(* IEC 61131-3 sources: lacyccom/src/Blocks/Drives (part 2) *)

(* ---- classRtcSinamics.st ---- *)
USING Siemens.Simatic.Clocks;
USING System.DateTime;

NAMESPACE Simatic.Ax.LAcycCom
    CLASS LAcycCom_classRtcSinamics
        VAR
            statrtcRealTimeSyncPING         : BOOL;
            statRetSetrtcRealTimeSyncPING   : BOOL;
            statRetResetrtcRealTimeSyncPING : BOOL;
            statrequestBuffer               : Resourcemanager;
            statWriteDrivePara              : LAcycCom_classWriteDriveSingleParams;
            statFBState                     : LAcycCom_ReadWriteStatus := LAcycCom_ReadWriteStatus#FB_IDLE;   // States in the function block state machine
            statFBSubState                  : LAcycCom_ReadWriteStatus := LAcycCom_ReadWriteStatus#FB_BUSY_PING;   // States in the function block during processing (busy state)
            statStatus                      : WORD := STATUS_NO_CALL;   // Static value for output status
            statStateNumber                 : LAcycCom_ReadWriteStatus;   // State of the FB when error occurred
            stathardwareId                  : HW_IO;
            statsystemDateTime              : LDATE_AND_TIME;
            statWritepara                   : LAcycCom_classWriteDriveSingleParams;
            statactmilisecond               : DWORD;
            statexternTime                  : BOOL;
            StatEnablePing                  : BOOL;
        END_VAR

        VAR CONSTANT
            STATUS_EXECUTION_FINISHED   : WORD := WORD#16#0000;   // Execution finished without errors
            STATUS_NO_CALL              : WORD := WORD#16#7000;   // No call of FB
            STATUS_ALLOCATE             : WORD := WORD#16#7001;   // FB is currently allocating a request element
            STATUS_GET_RESOURCE         : WORD := WORD#16#7002;   // FB is waiting until it has “speaking rights”
            STATUS_BUSY                 : WORD := WORD#16#7003;   // FB is currently in processing
            STATUS_RELEASE              : WORD := WORD#16#7004;   // FB is releasing the allocated element
            ERR_UNDEFINED_STATE         : WORD := WORD#16#8611;   // Error due to an undefined state
        END_VAR

        METHOD PUBLIC execute

            IF NOT (statFBState = LAcycCom_ReadWriteStatus#FB_IDLE OR
                statFBState = LAcycCom_ReadWriteStatus#FB_DONE OR
                statFBState = LAcycCom_ReadWriteStatus#FB_ERROR ) THEN  // Functionality running
                CASE statFBState OF
                    LAcycCom_ReadWriteStatus#FB_FIRST_CYCLE:  // First cycle state

                        This.FIRST_CYCLE();

                    LAcycCom_ReadWriteStatus#FB_BUSY:

                        This.BUSY();

                    ELSE
                    statStatus := ERR_UNDEFINED_STATE;
                    statStateNumber := statFBState;
                    statFBState := LAcycCom_ReadWriteStatus#FB_ERROR;
                END_CASE;
            END_IF;

        END_METHOD

        Method Private FIRST_CYCLE

            statrtcRealTimeSyncPING         := FALSE;
            statRetSetrtcRealTimeSyncPING   := FALSE;
            statRetResetrtcRealTimeSyncPING := FALSE;

            statFBState     := LAcycCom_ReadWriteStatus#FB_BUSY;
            statFBSubState  := LAcycCom_ReadWriteStatus#FB_BUSY_PING_RESET;
        END_METHOD

        Method PRIVATE Busy
            VAR
                actDays         : INT;
                actMonth        : INT;
                actYear         : INT;
                actHour         : INT;
                actMinute       : INT;
                actSecond       : INT;
                actMillisecond  : INT;
                elapsedYears    : INT;
                elapsedDays     : DINT;
                loop            : DINT;
            END_VAR

            CASE statFBSubState OF
                LAcycCom_ReadWriteStatus#FB_BUSY_PING_RESET:
                    IF statRetResetrtcRealTimeSyncPING THEN
                        statFBSubState := LAcycCom_ReadWriteStatus#FB_BUSY_WRREC;

                        statWriteDrivePara.execute();
                        statWriteDrivePara.Start(driveObjectId  := UINT#1,   // Optional: Identification number of the drive object (value =0: driveObjectId is NOT used, i.e. the corresponding drive object is only addressed via the hardwareId)
                                                hardwareId      := stathardwareId,   // Hardware identifier of the hardware module
                                                parameterNumber := UINT#3100,   // Number of the parameter
                                                index           := UINT#0,   // Parameter index
                                                value           := REAL#1.0,
                                                dwValue         := DWORD#0
                                                );
                    END_IF;

                LAcycCom_ReadWriteStatus#FB_BUSY_WRREC:
                    statWriteDrivePara.execute();

                    IF  statWriteDrivePara.Status() = LAcycComstateDef#DONE THEN
                        statFBSubState := LAcycCom_ReadWriteStatus#FB_BUSY_WRREC_1;
                        IF StatEnablePing THEN
                            statWriteDrivePara.Start(driveObjectId  := UINT#1,   // Optional: Identification number of the drive object (value =0: driveObjectId is NOT used, i.e. the corresponding drive object is only addressed via the hardwareId)
                                                    hardwareId      := stathardwareId,   // Hardware identifier of the hardware module
                                                    parameterNumber := UINT#3103,   // Number of the parameter
                                                    index           := UINT#0,   // Parameter index
                                                    value           := REAL#0.0,
                                                    dwValue         := DWORD#0
                                                    );
                        ELSE
                            statWriteDrivePara.Start(driveObjectId  := UINT#1,   // Optional: Identification number of the drive object (value =0: driveObjectId is NOT used, i.e. the corresponding drive object is only addressed via the hardwareId)
                                                    hardwareId      := stathardwareId,   // Hardware identifier of the hardware module
                                                    parameterNumber := UINT#3103,   // Number of the parameter
                                                    index           := UINT#0,   // Parameter index
                                                    value           := REAL#2.0,
                                                    dwValue         := DWORD#0
                                                    );
                        END_IF;
                    END_IF;

                LAcycCom_ReadWriteStatus#FB_BUSY_WRREC_1:
                    statWriteDrivePara.execute();

                    IF  statWriteDrivePara.Status() = LAcycComstateDef#DONE THEN
                        statFBSubState := LAcycCom_ReadWriteStatus#FB_BUSY_PING;
                    END_IF;

                LAcycCom_ReadWriteStatus#FB_BUSY_PING:
                    statrtcRealTimeSyncPING := StatEnablePing;
                    IF statRetSetrtcRealTimeSyncPING OR NOT StatEnablePing THEN

                        IF NOT statexternTime THEN
                            GetSystemDateTime(value => statsystemDateTime);
                        END_IF;

                        SplitDateAndTime(value := statsystemDateTime,
                        year => actYear,
                        month => actMonth,
                        day => actDays,
                        hour => actHour,
                        minute => actMinute,
                        second => actSecond,
                        millisecond => actMillisecond);

                        //add number of days from full years, subtracting the current year
                        FOR loop := 1992 TO (actYear - 1) DO
                            IF loop MOD 4 = 0 AND loop <> 2100 THEN
                                elapsedDays := elapsedDays + 366;
                            ELSE
                                elapsedDays := elapsedDays + 365;
                            END_IF;
                        END_FOR;

                        //add days from full months of the current year
                        IF actMonth > 1 THEN
                            elapsedDays := elapsedDays + 31;
                        END_IF;
                        IF actMonth > 2 THEN
                            IF actYear MOD 4 = 0 AND NOT (actYear = 2100) THEN
                                elapsedDays := elapsedDays + 29;
                            ELSE
                                elapsedDays := elapsedDays + 28;
                            END_IF;
                        END_IF;
                        IF actMonth > 3 THEN
                            elapsedDays := elapsedDays + 31;
                        END_IF;
                        IF actMonth > 4 THEN
                            elapsedDays := elapsedDays + 30;
                        END_IF;
                        IF actMonth > 5 THEN
                            elapsedDays := elapsedDays + 31;
                        END_IF;
                        IF actMonth > 6 THEN
                            elapsedDays := elapsedDays + 30;
                        END_IF;
                        IF actMonth > 7 THEN
                            elapsedDays := elapsedDays + 31;
                        END_IF;
                        IF actMonth > 8 THEN
                            elapsedDays := elapsedDays + 31;
                        END_IF;
                        IF actMonth > 9 THEN
                            elapsedDays := elapsedDays + 30;
                        END_IF;
                        IF actMonth > 10 THEN
                            elapsedDays := elapsedDays + 31;
                        END_IF;
                        IF actMonth > 11 THEN
                            elapsedDays := elapsedDays + 30;
                        END_IF;

                        //add days from current month
                        elapsedDays := elapsedDays + actDays;
                        statactmilisecond :=TO_DWORD (TO_UDINT(actMillisecond) + UDINT#1000 * (TO_UDINT(actSecond) + UDINT#60 * (TO_UDINT(actMinute + 60 * ( actHour)))));

                        statFBSubState := LAcycCom_ReadWriteStatus#FB_BUSY_WRREC_2;
                        statWriteDrivePara.execute();
                        statWriteDrivePara.Start(driveObjectId  := UINT#1,   // Optional: Identification number of the drive object (value =0: driveObjectId is NOT used, i.e. the corresponding drive object is only addressed via the hardwareId)
                                                hardwareId      := stathardwareId,   // Hardware identifier of the hardware module
                                                parameterNumber := UINT#3101,   // Number of the parameter
                                                index           := UINT#1,   // Parameter index
                                                value           := TO_REAL(elapsedDays+8034),
                                                dwValue         := DWORD#0
                                                );
                    END_IF;

                LAcycCom_ReadWriteStatus#FB_BUSY_WRREC_2 :
                    statWriteDrivePara.execute();

                    IF  statWriteDrivePara.Status() = LAcycComstateDef#DONE THEN

                        statFBSubState := LAcycCom_ReadWriteStatus#FB_BUSY_WRREC_3;
                        statWriteDrivePara.execute();
                        statWriteDrivePara.Start(driveObjectId  := UINT#1,   // Optional: Identification number of the drive object (value =0: driveObjectId is NOT used, i.e. the corresponding drive object is only addressed via the hardwareId)
                                                hardwareId      := stathardwareId,   // Hardware identifier of the hardware module
                                                parameterNumber := UINT#3101,   // Number of the parameter
                                                index           := UINT#0,   // Parameter index
                                                value           := REAL#0.0,
                                                dwValue         := statactmilisecond

                                        );

                    END_IF;

                LAcycCom_ReadWriteStatus#FB_BUSY_WRREC_3 :
                    statWriteDrivePara.execute();
                    IF  statWriteDrivePara.Status() = LAcycComstateDef#DONE THEN
                            statFBState             := LAcycCom_ReadWriteStatus#FB_DONE;
                            statrtcRealTimeSyncPING := FALSE;
                    END_IF;
            END_CASE;

        END_METHOD

        METHOD PUBLIC Start : BOOL
            VAR_INPUT
                hardwareId      : HW_IO;
                enablePingSnap  : BOOL := TRUE;
            END_VAR
                         // starts functionality
             IF NOT ((statFBState = LAcycCom_ReadWriteStatus#FB_IDLE OR
                    statFBState = LAcycCom_ReadWriteStatus#FB_DONE OR
                    statFBState = LAcycCom_ReadWriteStatus#FB_ERROR) AND
                    statrequestBuffer <> NULL) THEN
                        Start := FALSE;
             ELSE
               // Initialisation
                        StatEnablePing  := enablePingSnap;
                        Start           := TRUE;
                        statexternTime  := FALSE;
                        stathardwareId  := hardwareId;
                        statFBState     := LAcycCom_ReadWriteStatus#FB_FIRST_CYCLE;

             END_IF;

            statWriteDrivePara.Config(requestBuffer := statrequestBuffer);
        end_METHOD

        METHOD PUBLIC StartTimeSet : BOOL
            VAR_INPUT
                hardwareId : HW_IO;
                enablePingSnap  : BOOL := FALSE;
                SetTime : LDATE_AND_TIME;
            END_VAR
                         // starts functionality
             IF NOT ((statFBState = LAcycCom_ReadWriteStatus#FB_IDLE OR
                    statFBState = LAcycCom_ReadWriteStatus#FB_DONE OR
                    statFBState = LAcycCom_ReadWriteStatus#FB_ERROR) AND
                    statrequestBuffer <> NULL) THEN
                    StartTimeSet := FALSE;
             ELSE
               // Initialisation
                    StatEnablePing      := enablePingSnap;
                    StartTimeSet        := TRUE;
                    statexternTime      := TRUE;
                    stathardwareId      := hardwareId;
                    statsystemDateTime  := SetTime;
                    statFBState         := LAcycCom_ReadWriteStatus#FB_FIRST_CYCLE;
             END_IF;

            statWriteDrivePara.Config(requestBuffer := statrequestBuffer);
        end_METHOD

        METHOD PUBLIC getPing : BOOL
            getPing := statrtcRealTimeSyncPING;
            IF statrtcRealTimeSyncPING THEN
                statRetSetrtcRealTimeSyncPING := TRUE;
                statRetResetrtcRealTimeSyncPING := FALSE;
            ELSE
                statRetSetrtcRealTimeSyncPING := FALSE;
                statRetResetrtcRealTimeSyncPING := TRUE;
            END_IF;
        end_METHOD

        METHOD PUBLIC Config : BOOL
            VAR_INPUT
                requestBuffer : Resourcemanager;   // Connection to the request buffer of the resource manager. All LAcycCom blocks have to use the same request buffer
             END_VAR

             statrequestBuffer := requestBuffer;

        END_METHOD

        METHOD PUBLIC Status   : LAcycComstateDef;
            CASE statFBState OF
                LAcycCom_ReadWriteStatus#FB_IDLE:
                    Status := LAcycComstateDef#IDLE;

                LAcycCom_ReadWriteStatus#FB_FIRST_CYCLE,
                LAcycCom_ReadWriteStatus#FB_ALLOCATE,
                LAcycCom_ReadWriteStatus#FB_GET_RESOURCE,
                LAcycCom_ReadWriteStatus#FB_BUSY,
                LAcycCom_ReadWriteStatus#FB_RELEASE:
                    Status := LAcycComstateDef#BUSY;

                LAcycCom_ReadWriteStatus#FB_DONE:
                    Status := LAcycComstateDef#DONE;

                LAcycCom_ReadWriteStatus#FB_ERROR:
                    Status := LAcycComstateDef#Error;

            ELSE
                ;
            END_CASE;
        END_METHOD

        METHOD PUBLIC diag : LAcycCom_ooptypeDrivediagnostics
            diag := statWriteDrivePara.errordiagnostics();
        END_METHOD

    END_CLASS

END_NAMESPACE

(* ---- classWriteDriveParams.st ---- *)
using System.Timer;
using siemens.Simatic.DistributedIO;

NAMESPACE Simatic.Ax.LAcycCom
    CLASS LAcycCom_classWriteDriveParams EXTENDS ReadWriteParameter
        VAR PRIVATE
            statparameterCount   : INT := -1;
            dataset              : Array[0..LAcycComConstantsInt#LACYCCOM_WRITE_PARAMETERS_UPPER_LIM] of LAcycCom_typeDriveDataset;          // Dataset with all parameters to be read
            statReqWriteParameter: LAcycCom_TypestatReqWriteParameter;                                                                       // Request telegram to change the parameter values
            statReqReadParameter : LAcycCom_TypestatstatReqParameter;                                                                        // Request telegram
            statParameter        : Array[0..LAcycComConstantsInt#LACYCCOM_WRITE_PARAMETERS_UPPER_LIM] of LAcycCom_TypestatstatParameter;     // Parameter dataset
            parameterAddress     : Array[0..LAcycComConstantsInt#LACYCCOM_WRITE_PARAMETERS_UPPER_LIM] of LAcycCom_TypestatparameterAddress;  // Parameter data in telegram
        END_VAR

        VAR CONSTANT
          WRITE_PARAMETERS_UPPER_LIM : INT := 18;   // Maximum count of parameters
          LENGTH_WRITE_TELEGRAM_UPPER_LIM : INT := 227;   // Maximum length of parameter information when using WRREC
        END_VAR

        METHOD OVERRIDE BUSY
            VAR_TEMP
                tempCmdValid         : BOOL;                       // TRUE: New data record was received and is valid
                tempStatusWord       : WORD;                       // Temporary status
                tempWord             : WORD;                       // Temporary WORD variable
                tempPointer          : INT;                        // Temporary pointer variable
                tempLoopIndex        : INT;                        // Temporary loop index variable
                tempBlkVariant       : INT;                        // Temporary result of MOVE_BLK_VARIANT
                tempCmdStatus        : DWORD;                      // Temporary status of WRREC and RDREC command
                tempDWord            : DWORD;                      // Temporary DWORD variable
                tempVoidHeader       : LAcycCom_Typestatheader;    // Temporary empty header structure
                tempActualElementReal: LAcycCom_typeDriveDataset;  // Temporary element of the dataset (REAL values)
             END_VAR
             IF (statrequestBuffer.GetRessource(statAllocatedIndex) = LAcycCom_ResourceManagerRetval#STATUS_BUSY) THEN
                CASE statFBSubState OF
                    LAcycCom_ReadWriteStatus#FB_GET_SUBSTATE:
                      statFBSubState := LAcycCom_ReadWriteStatus#FB_BUSY_WRREC_1;

                      // Clearing the sending write buffer
                      statReqWriteParameter.header := tempVoidHeader;
                      FOR tempLoopIndex := 0 TO LENGTH_WRITE_TELEGRAM_UPPER_LIM DO
                      statReqWriteParameter.data[tempLoopIndex] := BYTE#16#00;
                      END_FOR;

                      FOR tempLoopIndex := 0 TO LENGTH_WRITE_TELEGRAM_UPPER_LIM DO
                         THIS.atmpRec[tempLoopIndex] := BYTE#0;
                      END_FOR;

                    LAcycCom_ReadWriteStatus#FB_BUSY_WRREC_1, LAcycCom_ReadWriteStatus#FB_BUSY_WRREC_2:  // Writing the dataset configuration into the drive object

                    IF (statCmdBusy = FALSE) AND (statFBSubState = LAcycCom_ReadWriteStatus#FB_BUSY_WRREC_1) AND  NOT(statFBState = LAcycCom_ReadWriteStatus#FB_ERROR) THEN
                      // Resets WRREC command
                      instWRREC(request := FALSE,
                      RECORD := THIS.atmpRec);

                      // Creating header data
                     statReqReadParameter.header.refNo := statRefNo; // Telegram reference number
                     statReqReadParameter.header.reqId := BYTE#16#01;  // 0x01 = request parameters
                     statReqReadParameter.header.doId := TO_BYTE(statDoId);  // Drive object identification number
                     statReqReadParameter.header.parameterNo := TO_BYTE(statCountOfElements);  // Count of parameters

                      // Copying the dataset into a static variable (depending on the used PLC data type)

                        FOR tempLoopIndex := 0 TO statCountOfElements - 1 BY 1 DO
                         tempActualElementReal:= dataset[tempLoopIndex];
                         statParameter[tempLoopIndex].index := UINT#0;
                         statParameter[tempLoopIndex].parameterNo := tempActualElementReal.parameterNumber;
                         statParameter[tempLoopIndex].realValue := tempActualElementReal.Rvalue;
                         statParameter[tempLoopIndex].dwordValue := tempActualElementReal.DWvalue;
                         statReqReadParameter.parameterAddress[tempLoopIndex].parameterNo := statParameter[tempLoopIndex].parameterNo;  // Parameter number
                         statReqReadParameter.parameterAddress[tempLoopIndex].index := statParameter[tempLoopIndex].index;  // Subindex of parameter
                        END_FOR;

                    ELSIF (statCmdBusy = FALSE) AND (statFBSubState = LAcycCom_ReadWriteStatus#FB_BUSY_WRREC_2) AND  NOT(statFBState = LAcycCom_ReadWriteStatus#FB_ERROR) THEN
                      // Resets WRREC command
                      instWRREC(request := FALSE,
                                 RECORD := THIS.atmpRec);

                       tempPointer := 0;
                      // Creating header data
                     statReqWriteParameter.header.refNo := statRefNo; // Telegram reference number
                     statReqWriteParameter.header.reqId := BYTE#16#02;  // 0x02 = change parameters
                     statReqWriteParameter.header.doId := TO_BYTE(statDoId);  // Drive object identification number
                     statReqWriteParameter.header.parameterNo := TO_BYTE(statCountOfElements);  // Count of parameters

                      FOR tempLoopIndex := 0 TO statCountOfElements - 1 BY 1 DO
                       statReqWriteParameter.data [tempPointer] := BYTE#16#10; // Attribute of parameters (0x10=Value, 0x30=Text)
                       statReqWriteParameter.data [tempPointer + 1] := BYTE#16#01; // No. of elements (for single elements=1)

                        // Parameter number
                       statReqWriteParameter.data [tempPointer + 3] := statParameter[tempLoopIndex].parameterNo.%B0;
                       statReqWriteParameter.data [tempPointer + 2] := statParameter[tempLoopIndex].parameterNo.%B1;

                        // Subindex of parameter
                       statReqWriteParameter.data [tempPointer + 5] := statParameter[tempLoopIndex].index.%B0;
                       statReqWriteParameter.data [tempPointer + 4] := statParameter[tempLoopIndex].index.%B1;

                        // Points to the next parameter address
                         tempPointer := tempPointer + 6;
                      END_FOR;

                      // Creating parameter address
                      FOR tempLoopIndex := 0 TO statCountOfElements - 1 BY 1 DO

                        IF (statParameter[tempLoopIndex].format = FORMAT_ERROR) THEN
                         statParameter[tempLoopIndex].format := TO_BYTE(FORMAT_FLOATING_POINT);
                        END_IF;

                       statReqWriteParameter.data [tempPointer] := statParameter[tempLoopIndex].format; // Format of parameter
                       statReqWriteParameter.data [tempPointer + 1] := BYTE#16#01; // Count of values

                        CASE TO_SINT(statParameter[tempLoopIndex].format) OF
                          FORMAT_INTEGER_8:
                            IF NOT (statParameter[tempLoopIndex].realValue = 0.0) THEN
                               tempDWord := TO_DWORD(TO_SINT(statParameter[tempLoopIndex].realValue));

                            ELSE
                               tempDWord := statParameter[tempLoopIndex].dwordValue;
                            END_IF;

                           statReqWriteParameter.data [tempPointer + 3] := tempDWord.%B1;
                           statReqWriteParameter.data [tempPointer + 2] := tempDWord.%B0;
                             tempPointer := tempPointer + 4;  // Points to the next parameter address

                          FORMAT_INTEGER_16:
                            IF NOT (statParameter[tempLoopIndex].realValue = 0.0) THEN
                               tempDWord := TO_DWORD(TO_DINT(statParameter[tempLoopIndex].realValue));

                            ELSE
                               tempDWord := statParameter[tempLoopIndex].dwordValue;
                            END_IF;

                           statReqWriteParameter.data [tempPointer + 3] := tempDWord.%B0;
                           statReqWriteParameter.data [tempPointer + 2] := tempDWord.%B1;
                             tempPointer := tempPointer + 4;  // Points to the next parameter address

                          FORMAT_INTEGER_32:
                            IF NOT (statParameter[tempLoopIndex].realValue = 0.0) THEN
                               tempDWord := TO_DWORD(TO_DINT(statParameter[tempLoopIndex].realValue));

                            ELSE
                               tempDWord := statParameter[tempLoopIndex].dwordValue;
                            END_IF;

                           statReqWriteParameter.data [tempPointer + 5] := tempDWord.%B0;
                           statReqWriteParameter.data [tempPointer + 4] := tempDWord.%B1;
                           statReqWriteParameter.data [tempPointer + 3] := tempDWord.%B2;
                           statReqWriteParameter.data [tempPointer + 2] := tempDWord.%B3;

                             tempPointer := tempPointer + 6; // Points to the next parameter address

                          FORMAT_UNSIGNED_8, FORMAT_OCTET_STRING: // V1.5 change OCTET_STRING:
                            IF NOT (statParameter[tempLoopIndex].realValue = 0.0) THEN
                               tempDWord := TO_DWORD(TO_USINT(statParameter[tempLoopIndex].realValue));

                            ELSE
                               tempDWord := statParameter[tempLoopIndex].dwordValue;
                            END_IF;

                           statReqWriteParameter.data [tempPointer + 3] := tempDWord.%B1;
                           statReqWriteParameter.data [tempPointer + 2] := tempDWord.%B0;
                             tempPointer := tempPointer + 4;  // Points to the next parameter address

                          FORMAT_UNSIGNED_16:
                            IF NOT (statParameter[tempLoopIndex].realValue = 0.0) THEN
                               tempDWord := TO_DWORD(TO_UDINT(statParameter[tempLoopIndex].realValue));

                            ELSE
                               tempDWord := statParameter[tempLoopIndex].dwordValue;
                            END_IF;

                           statReqWriteParameter.data [tempPointer + 3] := tempDWord.%B0;
                           statReqWriteParameter.data [tempPointer + 2] := tempDWord.%B1;
                             tempPointer := tempPointer + 4;  // Points to the next parameter address

                          FORMAT_UNSIGNED_32, FORMAT_TIME_DIFFERENCE:
                            IF NOT (statParameter[tempLoopIndex].realValue = 0.0) THEN
                               tempDWord := TO_DWORD(TO_UDINT(statParameter[tempLoopIndex].realValue));

                            ELSE
                               tempDWord := statParameter[tempLoopIndex].dwordValue;
                            END_IF;

                           statReqWriteParameter.data [tempPointer + 5] := tempDWord.%B0;
                           statReqWriteParameter.data [tempPointer + 4] := tempDWord.%B1;
                           statReqWriteParameter.data [tempPointer + 3] := tempDWord.%B2;
                           statReqWriteParameter.data [tempPointer + 2] := tempDWord.%B3;

                             tempPointer := tempPointer + 6; // Points to the next parameter address
                          FORMAT_FLOATING_POINT, FORMAT_DOUBLE_WORD:
                            IF NOT (statParameter[tempLoopIndex].realValue = 0.0) THEN
                               tempDWord := TO_DWORD(statParameter[tempLoopIndex].realValue);

                            ELSE
                               tempDWord := statParameter[tempLoopIndex].dwordValue;
                            END_IF;

                           statReqWriteParameter.data [tempPointer + 5] := tempDWord.%B0;
                           statReqWriteParameter.data [tempPointer + 4] := tempDWord.%B1;
                           statReqWriteParameter.data [tempPointer + 3] := tempDWord.%B2;
                           statReqWriteParameter.data [tempPointer + 2] := tempDWord.%B3;

                             tempPointer := tempPointer + 6;  // Points to the next parameter address
                          FORMAT_BYTE:
                            IF NOT (statParameter[tempLoopIndex].realValue = 0.0) THEN
                               tempDWord := TO_DWORD(statParameter[tempLoopIndex].realValue);

                            ELSE
                               tempDWord := statParameter[tempLoopIndex].dwordValue;
                            END_IF;

                           statReqWriteParameter.data [tempPointer + 3] := tempDWord.%B1;
                           statReqWriteParameter.data [tempPointer + 2] := tempDWord.%B0;
                             tempPointer := tempPointer + 4;  // Points to the next parameter address

                          FORMAT_WORD:
                            IF NOT (statParameter[tempLoopIndex].realValue = 0.0) THEN
                               tempDWord := TO_DWORD(statParameter[tempLoopIndex].realValue);

                            ELSE
                               tempDWord := statParameter[tempLoopIndex].dwordValue;
                            END_IF;

                           statReqWriteParameter.data [tempPointer + 3] := tempDWord.%B0;
                           statReqWriteParameter.data [tempPointer + 2] := tempDWord.%B1;
                             tempPointer := tempPointer + 4;  // Points to the next parameter address

                          ELSE
                            ;
                        END_CASE;
                      END_FOR; // // Creating parameter address
                    END_IF; // statCmdBusy = FALSE AND statParameterConfig = TRUE

                    SerializeBig(UINT#0,
                    statReqReadParameter,
                    THIS.atmpSend );

                    IF (statFBSubState = LAcycCom_ReadWriteStatus#FB_BUSY_WRREC_1) AND  NOT(statFBState = LAcycCom_ReadWriteStatus#FB_ERROR) THEN
                      SerializeBig(UINT#0,
                        statReqReadParameter,
                        THIS.atmpSend );
                      // WRREC command
                      instWRREC(REQUEST := TRUE,                                                // Transfer data record
                                 hardwareID := statHwId,           // ID number of the hardware component
                                 INDEX  := statDataRecordNo,   // Data record number
                                 LENGTH := UINT#0,             // Maximum length of the data record to be transferred in bytes
                                 DONE   => statCmdDone,        // Data record was transferred
                                 BUSY   => statCmdBusy,        // The writing process is NOT yet complete
                                 ERROR  => statCmdError,       // An error occurred during the writing process
                                 STATUS =>  tempCmdStatus,     // Status[1] = Error => Status[2] Error Decode + Status[3] Error Code
                                 RECORD := THIS.atmpSend);     // Data record

                    ELSIF (statFBSubState = LAcycCom_ReadWriteStatus#FB_BUSY_WRREC_2) AND  NOT(statFBState = LAcycCom_ReadWriteStatus#FB_ERROR) THEN
                      SerializeBig(UINT#0,
                        statReqWriteParameter,
                        THIS.atmpSend );
                        // WRREC command
                      instWRREC(REQUEST := TRUE,                                                // Transfer data record
                                 hardwareID := statHwId,           // ID number of the hardware component
                                 INDEX  := statDataRecordNo,   // Data record number
                                 LENGTH := UINT#0,             // Maximum length of the data record to be transferred in bytes
                                 DONE   => statCmdDone,        // Data record was transferred
                                 BUSY   => statCmdBusy,        // The writing process is NOT yet complete
                                 ERROR  => statCmdError,       // An error occurred during the writing process
                                 STATUS =>  tempCmdStatus,     // Status[1] = Error => Status[2] Error Decode + Status[3] Error Code
                                 RECORD := THIS.atmpSend);     // Data record
                    END_IF;

                    // Error occurred
                    IF (statCmdError = TRUE) AND  NOT(statFBState = LAcycCom_ReadWriteStatus#FB_ERROR) THEN
                      // Get the error information from the status information
                       tempStatusWord.%B0 := tempCmdStatus.%B1;
                       tempStatusWord.%B1 := tempCmdStatus.%B2;

                      // Temporary command status (80A1, 80A7, 80B5, 80C0, 80C1, 80C2, 80C3 oder 80C4) are valid and retry command
                      IF (tempStatusWord = WORD#16#80A1) OR  // Negative acknowledgment when writing to the module
                        (tempStatusWord = WORD#16#80A7) OR   // DP slave OR module is occupied (temporary error)
                        (tempStatusWord = WORD#16#80B5) OR   // DP slave OR module NOT ready
                        (tempStatusWord = WORD#16#80C0) OR   // The data can only be written when the CPU is in STOP mode. Note: this means that writing by the user program is NOT possible. You can only write the data online with PG/PC.
                        (tempStatusWord = WORD#16#80C1) OR   // The data of the previous write job on the module for the same data record have NOT yet been processed by the module.
                        (tempStatusWord = WORD#16#80C2) OR   // The module is currently processing the maximum possible number of jobs for a CPU.
                        (tempStatusWord = WORD#16#80C3) OR   // The required operating resources are currently occupied.
                        (tempStatusWord = WORD#16#80C4) THEN // Internal temporary error. Job could NOT be executed. Repeat the job. IF this error occurs often, check your installation for sources of electrical interference.

                        IF (statErrorCount >= MAX_ERROR_COUNT) THEN
                         statStateNumber := statFBSubState;
                         statSubfunctionStatus := tempStatusWord;
                         statStatus := ERR_WRREC_TEMP_COUNTER;
                         statFBState := LAcycCom_ReadWriteStatus#FB_ERROR;
                        ELSE
                         statErrorCount := statErrorCount + UINT#1;  // Increment internal error counter
                         statFBSubStateOld := statFBSubState;
                         statFBSubState := LAcycCom_ReadWriteStatus#FB_BUSY_WAIT;
                        END_IF;
                      ELSE
                       statStateNumber := statFBSubState;
                       statSubfunctionStatus := tempStatusWord;
                       statStatus := ERR_WRREC;
                       statFBState := LAcycCom_ReadWriteStatus#FB_ERROR;
                      END_IF; // Temporary command status (80A1, 80A7, 80B5, 80C0, 80C1, 80C2, 80C3 oder 80C4) are valid and retry command

                    ELSIF (statCmdBusy = FALSE) AND (statCmdDone = TRUE) AND  NOT(statFBState = LAcycCom_ReadWriteStatus#FB_ERROR) AND (statFBSubState = LAcycCom_ReadWriteStatus#FB_BUSY_WRREC_1) THEN  // Processing completed without errors
                     statErrorCount := UINT#0;  // V1.5.1 Reset error counter
                     statFBSubState := LAcycCom_ReadWriteStatus#FB_BUSY_RDREC_1; // WRREC completed and continue with RDREC

                    ELSIF (statCmdBusy = FALSE) AND (statCmdDone = TRUE) AND  NOT(statFBState = LAcycCom_ReadWriteStatus#FB_ERROR) AND (statFBSubState = LAcycCom_ReadWriteStatus#FB_BUSY_WRREC_2) THEN  // Processing completed without errors
                     statErrorCount := UINT#0;  // V1.5.1 Reset error counter
                     statFBSubState := LAcycCom_ReadWriteStatus#FB_BUSY_RDREC_2; // WRREC completed and continue with RDREC
                      // Clearing the receive buffer
                     statRespParameter.header := tempVoidHeader;
                      FOR tempLoopIndex := 0 TO LENGTH_READ_TELEGRAM_UPPER_LIM DO
                       statRespParameter.data[tempLoopIndex] := BYTE#16#00;
                      END_FOR;
                    END_IF; // statCmdError = TRUE

                    LAcycCom_ReadWriteStatus#FB_BUSY_RDREC_1, LAcycCom_ReadWriteStatus#FB_BUSY_RDREC_2:  // Reading the values from the drive object

                    // Resets RDREC command
                    IF (statCmdBusy = FALSE) THEN
                      instRDREC(request := FALSE,
                                 RECORD := THIS.atmpRec);

                    END_IF;

                    instRDREC(request := TRUE,                                                 // Transfer data record
                               hardwareID := statHwId,           // ID number of the hardware component
                               INDEX     := statDataRecordNo,   // Data record number
                               MAXLENGTH := UINT#0,             // Maximum length in bytes of the data record information to be read
                               VALID     =>  tempCmdValid,      // New data record was received and is valid
                               BUSY      => statCmdBusy,        // The reading process is NOT yet complete
                               ERROR     => statCmdError,       // An error occurred during the reading process
                               STATUS    =>  tempCmdStatus,     // Status[1] = Error => Status[2] Error Decode + Status[3] Error Code
                               RECORD    := THIS.atmpRec);      // Destination area for the data record read

                    DeserializeBig(UINT#0,
                                THIS.atmpRec,
                                statRespParameter);

                    // Error occurred
                    IF (statCmdError = TRUE) AND  NOT(statFBState = LAcycCom_ReadWriteStatus#FB_ERROR) THEN
                      // Get the error information from the status information
                       tempStatusWord.%B0 := tempCmdStatus.%B1;
                       tempStatusWord.%B1 := tempCmdStatus.%B2;

                      // Temporary command status (80A0, 80A7, 80B5, 80C0, 80C1, 80C2, 80C3 oder 80C4) are valid and retry command
                      IF (tempStatusWord = WORD#16#80A0) OR  // Negative acknowledgment when reading the module
                        (tempStatusWord = WORD#16#80A7) OR   // DP slave OR module is occupied (temporary error)
                        (tempStatusWord = WORD#16#80B5) OR   // DP slave OR module NOT ready
                        (tempStatusWord = WORD#16#80C0) OR   // The data can only be written when the CPU is in STOP mode. Note: this means that writing by the user program is NOT possible. You can only write the data online with PG/PC.
                        (tempStatusWord = WORD#16#80C1) OR   // The data of the previous write job on the module for the same data record have NOT yet been processed by the module.
                        (tempStatusWord = WORD#16#80C2) OR   // The module is currently processing the maximum possible number of jobs for a CPU.
                        (tempStatusWord = WORD#16#80C3) OR   // The required operating resources are currently occupied.
                        (tempStatusWord = WORD#16#80C4) THEN // Internal temporary error. Job could NOT be executed. Repeat the job. IF this error occurs often, check your installation for sources of electrical interference.

                        IF (statErrorCount >= MAX_ERROR_COUNT) THEN

                         statStateNumber := statFBSubState;
                         statSubfunctionStatus := tempStatusWord;
                         statStatus := ERR_RDREC_TEMP_COUNTER;
                         statFBState := LAcycCom_ReadWriteStatus#FB_ERROR;
                        ELSE
                         statErrorCount := statErrorCount + UINT#1;  // Increment internal error counter
                         statFBSubStateOld := statFBSubState;
                          // V1.3.2. IF error 80A0 THEN should be retry with WRREC command
                          IF (tempStatusWord = WORD#16#80A0) AND statFBSubState = LAcycCom_ReadWriteStatus#FB_BUSY_RDREC_1 THEN
                           statFBSubStateOld := LAcycCom_ReadWriteStatus#FB_BUSY_WRREC_1;
                          ELSIF (tempStatusWord = WORD#16#80A0) AND statFBSubState = LAcycCom_ReadWriteStatus#FB_BUSY_RDREC_2 THEN
                           statFBSubStateOld := LAcycCom_ReadWriteStatus#FB_BUSY_WRREC_2;
                          END_IF;
                         statFBSubState := LAcycCom_ReadWriteStatus#FB_BUSY_WAIT;
                        END_IF;
                      ELSE

                       statStateNumber := statFBSubState;
                       statSubfunctionStatus := tempStatusWord;
                       statStatus := ERR_RDREC;
                       statFBState := LAcycCom_ReadWriteStatus#FB_ERROR;
                      END_IF; // Temporary command status (80A0, 80A7, 80B5, 80C0, 80C1, 80C2, 80C3 oder 80C4) are valid and retry command

                      // Error : Reference number of the request does NOT match with the response reference number
                    ELSIF (statCmdBusy = FALSE) AND
                      (statRefNo <> statRespParameter.header.refNo) AND
                      (tempCmdValid = TRUE) THEN

                     statStateNumber := statFBSubState;
                     statStatus := ERR_REFERENCE_NO;
                     statFBState := LAcycCom_ReadWriteStatus#FB_ERROR;

                      // Error : Invalid response from the drive object (reqId: 16#01 - reading parameter successful; 16#81: reading parameter finished with error; 16#02: writing parameter sucessful; 16#82: writing parameter finished with error)
                    ELSIF (statCmdBusy = FALSE) AND
                      NOT (statRespParameter.header.reqId = BYTE#16#81 OR statRespParameter.header.reqId = BYTE#16#01 OR statRespParameter.header.reqId = BYTE#16#02 OR statRespParameter.header.reqId = BYTE#16#82) AND
                      (tempCmdValid = TRUE) THEN

                     statStateNumber := statFBSubState;
                     statStatus := ERR_RESPONSE_ID;
                     statFBState := LAcycCom_ReadWriteStatus#FB_ERROR;

                      // Error : The received number of parameters does NOT match with the requested number of parameters
                    ELSIF (statCmdBusy = FALSE) AND
                      (statCountOfElements <> TO_INT(statRespParameter.header.parameterNo)) AND
                      (tempCmdValid = TRUE) THEN

                     statStateNumber := statFBSubState;
                     statStatus := ERR_PARAMETER_NO;
                     statFBState := LAcycCom_ReadWriteStatus#FB_ERROR;

                      // Error : The drive object does NOT match with the responsed DO
                    ELSIF (statCmdBusy = FALSE) AND
                      (TO_BYTE(statDoId) <> statRespParameter.header.doId) AND
                      (tempCmdValid = TRUE) THEN

                     statStateNumber := statFBSubState;
                     statStatus := ERR_DRIVE_OBJECT_NO;
                     statFBState := LAcycCom_ReadWriteStatus#FB_ERROR;

                      // No error occurred during reading parameters
                    ELSIF (statCmdBusy = FALSE) AND (tempCmdValid = TRUE) AND  NOT(statFBState = LAcycCom_ReadWriteStatus#FB_ERROR) THEN

                      IF (statFBSubState = LAcycCom_ReadWriteStatus#FB_BUSY_RDREC_1) THEN

                        // Analyse of the response buffer
                         tempPointer := 0;
                        FOR tempLoopIndex := 0 TO statCountOfElements - 1 DO
                         statParameter[tempLoopIndex].format := statRespParameter.data [tempPointer];  // Format of the parameter

                          // Format = Error
                          IF (((TO_SINT(statRespParameter.data [tempPointer]) > FORMAT_DOUBLE_WORD) OR
                            ((TO_SINT(statRespParameter.data [tempPointer]) > FORMAT_FLOATING_POINT) AND (TO_SINT(statRespParameter.data [tempPointer]) < FORMAT_OCTET_STRING)) OR
                            ((TO_SINT(statRespParameter.data [tempPointer]) > FORMAT_OCTET_STRING) AND (TO_SINT(statRespParameter.data [tempPointer]) < FORMAT_TIME_DIFFERENCE)) OR
                            ((TO_SINT(statRespParameter.data [tempPointer]) > FORMAT_TIME_DIFFERENCE) AND (TO_SINT(statRespParameter.data [tempPointer]) < FORMAT_BYTE)) OR
                            (TO_SINT(statRespParameter.data [tempPointer]) < FORMAT_INTEGER_8))) AND (TO_SINT(statRespParameter.data [tempPointer]) <> FORMAT_ZERO)
                          THEN

                           statParameter[tempLoopIndex].errorValue := statRespParameter.data [tempPointer + 3];
                            // Points to the next parameter address
                             tempPointer := tempPointer + 6;

                          ELSE
                            CASE TO_SINT(statRespParameter.data [tempPointer]) OF
                              FORMAT_INTEGER_8, FORMAT_UNSIGNED_8, FORMAT_BYTE, FORMAT_INTEGER_16, FORMAT_UNSIGNED_16, FORMAT_OCTET_STRING, FORMAT_WORD:
                               statParameter[tempLoopIndex].errorValue := BYTE#16#FF; // Sets the error status and diagnostic
                                 tempPointer := tempPointer + 4; // Points to the next parameter address

                              FORMAT_INTEGER_32, FORMAT_UNSIGNED_32, FORMAT_TIME_DIFFERENCE, FORMAT_FLOATING_POINT, FORMAT_DOUBLE_WORD:
                               statParameter[tempLoopIndex].errorValue := BYTE#16#FF; // Sets the error status and diagnostics
                                 tempPointer := tempPointer + 6; // Points to the next parameter address

                              ELSE
                                ;
                            END_CASE;
                          END_IF; // Format = Error
                        END_FOR; // Analyse of the response buffer

                       statCmdBusy := FALSE;
                       statCmdError := FALSE;
                       statFBState := LAcycCom_ReadWriteStatus#FB_BUSY;
                       statFBSubState := LAcycCom_ReadWriteStatus#FB_BUSY_WRREC_2;
                      ELSE

                        // Error occurred during writing process (changing parameter values)
                        IF (statRespParameter.header.reqId = BYTE#16#82) THEN  // reqId: 16#82 (Error occurred during writing paramaters)
                           tempPointer := 0;

                          FOR tempLoopIndex := 0 TO statCountOfElements - 1 BY 1 DO
                            // Parameter error
                            IF (statRespParameter.data [tempPointer] = FORMAT_ERROR) THEN

                             statParameter[tempLoopIndex].errorValue := statRespParameter.data [tempPointer + 3]; // V1.3.2
                              // Save first parameter error in telegram
                              IF (statFirstParameterError = NO_PARAMETER_ERROR) THEN
                               statFirstParameterError := tempLoopIndex;
                                statdiagnostics.firstParameterError := statFirstParameterError;
                                statdiagnostics.errorValue := statParameter[tempLoopIndex].errorValue; // V1.3.2

                               statStateNumber := statFBSubState;
                               statStatus := ERR_PARAMETER;
                               statFBState := LAcycCom_ReadWriteStatus#FB_ERROR;
                              END_IF;

                               tempPointer := tempPointer + 6;  // Points to the next parameter address

                              // Parameter without errors
                            ELSE
                             statParameter[tempLoopIndex].errorValue := BYTE#16#FF;
                               tempPointer := tempPointer + 2;
                            END_IF;
                            dataset[tempLoopIndex]:=tempActualElementReal;
                          END_FOR;
                        END_IF; // Error occurred during writing process (changing parameter values)

                       statCmdBusy := FALSE;
                       statCmdError := FALSE;
                       statFBSubState := LAcycCom_ReadWriteStatus#FB_BUSY_WRREC_1;

                          // Next state is depending on the FB mode
                          IF NOT(statFBState = LAcycCom_ReadWriteStatus#FB_ERROR) THEN
                            statStatus := STATUS_RELEASE;
                            statFBState := LAcycCom_ReadWriteStatus#FB_RELEASE;

                          END_IF; // statMode = MODE_WITH_BUFFER_MANAGER
                      END_IF; // statParameterConfig = TRUE
                    END_IF; // statCmdError = TRUE

                    LAcycCom_ReadWriteStatus#FB_BUSY_WAIT:
                    // Timer for temporary errors
                    instIECTimer(signal := statTimerStart,
                    duration := TIMER_TEMP_ERROR);

                   statTimerStart := TRUE;
                    IF (instIECTimer.output = TRUE) THEN
                     statTimerStart := FALSE;
                     statFBSubState := statFBSubStateOld;
                    END_IF;

                  ELSE

                   statStatus := ERR_UNDEFINED_SUBSTATE;
                   statStateNumber := statFBState;
                   statFBState := LAcycCom_ReadWriteStatus#FB_ERROR;
                END_CASE;

              ELSE

               statStatus := ERR_COMMAND_TIMEOUT;
               statStateNumber := statFBState;
               statFBState := LAcycCom_ReadWriteStatus#FB_ERROR;
              END_IF; // ((buffer.element [statAllocatedIndex].enable = TRUE) AND (statMode = MODE_WITH_BUFFER_MANAGER)) OR statMode = MODE_WITHOUT_BUFFER_MANAGER

        END_METHOD

        //data type of driveobjectid has been changed from uint to int. This extra start method keeps compability to old versions of LAcycCom
        METHOD PUBLIC Start : BOOL
            VAR_INPUT
              driveObjectId : UINT;
              hardwareId    : HW_IO;
              parameterCount: INT := -1;
            END_VAR
            Start := THIS.Start(driveObjectId := TO_INT(driveObjectId), hardwareId := hardwareId, parameterCount := parameterCount);
          END_METHOD
          //data type of driveobjectid has been changed from uint to int. This extra start method can be used, if direct hw id is used and drive object is not used (equivalent to driveobjectid = -1)
          METHOD PUBLIC Start : BOOL
            VAR_INPUT
              hardwareId    : HW_IO;
              parameterCount: INT := -1;
          END_VAR
          Start := THIS.Start(driveObjectId := -1, hardwareId := hardwareId, parameterCount := parameterCount);
        END_METHOD

        METHOD PUBLIC Start : BOOL
            VAR_INPUT
                driveObjectId : INT := -1;  // Optional: Identification number of the drive object (value =-1: driveObjectId is NOT used, i.e. the corresponding drive object is only addressed via the hardwareId)
                hardwareId    : HW_IO;           // Hardware identifier of the hardware module
                parameterCount: INT := -1;       // Count of parameters to read (-1: read all parameter in dataset)
            END_VAR

             statparameterCount := parameterCount;
             statDoId := driveObjectId;
             statHwId := hardwareId;

             // starts functionality
             IF NOT ((statFBState = LAcycCom_ReadWriteStatus#FB_IDLE OR
                 statFBState = LAcycCom_ReadWriteStatus#FB_DONE OR
                 statFBState = LAcycCom_ReadWriteStatus#FB_ERROR) AND
                 statrequestBuffer <> NULL) THEN
                   Start := FALSE;
             ELSE
               // Initialisation
               Start := TRUE;
               statAllocatedIndex := -1;
               statSubfunctionStatus :=  WORD#16#0000;
               statDataRecordNo := DINT#0;
               statStateNumber := LAcycCom_ReadWriteStatus#FB_IDLE;
               statDatasetType := SINT#0;
               statFirstParameterError := -1;
               statErrorCount := UINT#0;
               statFBSubState := LAcycCom_ReadWriteStatus#FB_BUSY_WRREC;
               statFBState := LAcycCom_ReadWriteStatus#FB_FIRST_CYCLE;

               instIECTimer(signal := FALSE,
                             duration := TIMER_ALLOCATION);

             END_IF;
        END_METHOD

        METHOD PUBLIC DeleteList
            Var
                z : INT;
            END_VAR

            For z := 0 to LAcycComConstantsInt#LACYCCOM_WRITE_PARAMETERS_UPPER_LIM do
                dataset[z].DWvalue  := DWORD#0;
                dataset[z].errorValue := BYTE#0;
                dataset[z].index    := UINT#0;
                dataset[z].parameterNumber := UINT#0;
                dataset[z].Rvalue    := REAL#0.0;
            end_FOR;

            statCountOfElements := 0;

          END_METHOD

          METHOD PUBLIC AddatasetItem : INT //Rückgabewert = anzahl der Listeneinträge
            VAR_INPUT
                datasetItem : LAcycCom_typeDriveDataset;
                element_no  : INT := INT#-1; //-1 element an die liste anhängen. >=0 element überschreiben
            END_VAR

            IF element_no = -1 and statCountOfElements < LAcycComConstantsInt#LACYCCOM_WRITE_PARAMETERS_UPPER_LIM THEN
                    dataset[statCountOfElements] :=datasetItem;
                AddatasetItem := statCountOfElements;
                statCountOfElements := statCountOfElements + 1;

            ELSIF element_no > -1 and
                element_no < LAcycComConstantsInt#LACYCCOM_WRITE_PARAMETERS_UPPER_LIM and
                element_no <= statCountOfElements THEN
                    dataset[element_no] :=datasetItem;
                IF element_no = statCountOfElements THEN
                    statCountOfElements := statCountOfElements + 1;
                END_IF;
            ELSE
                AddatasetItem := -1;
            END_IF;

          END_METHOD

        METHOD PUBLIC ReaddatasetItem : LAcycCom_typeDriveDataset
          VAR_INPUT
              element_no  : INT := INT#0;
          END_VAR

          IF element_no >= 0 and element_no <= LAcycComConstantsInt#LACYCCOM_WRITE_PARAMETERS_UPPER_LIM THEN
              ReaddatasetItem := dataset[element_no];
          END_IF;

        END_METHOD

    END_CLASS
END_NAMESPACE

(* ---- classWriteDriveSingleParams.st ---- *)
using system.timer;
using siemens.Simatic.S71500.DistributedIO;

NAMESPACE Simatic.Ax.LAcycCom
    CLASS LAcycCom_classWriteDriveSingleParams EXTENDS ReadWriteParameter
        var Private
            statparameterNumber : UInt;   // Number of the parameter
            statindex : UInt;   // Parameter index
            statParameterValue : REAL;
            statParameterDWValue : DWORD;
            statReqWriteParameter  : LAcycCom_TypestatReqWriteParameter;   // Request telegram to change the parameter values
            statReqReadParameter   : LAcycCom_TypestatstatReqParameter;   // Request telegram
            statParameter   : Array[0..WRITE_PARAMETERS_UPPER_LIM] of LAcycCom_TypestatstatParameter;   // Parameter dataset
            parameterAddress   : Array[0..WRITE_PARAMETERS_UPPER_LIM] of LAcycCom_TypestatparameterAddress;   // Parameter data in telegram
        end_VAR

        VAR CONSTANT
         LENGTH_WRITE_TELEGRAM_UPPER_LIM : Int := 227;   // Maximum length of parameter information when using WRREC
         WRITE_PARAMETERS_UPPER_LIM : int := 0;
       end_var

        METHOD OVERRIDE BUSY
            VAR_TEMP
                tempCmdValid : Bool;   // TRUE: New data record was received and is valid
                tempStatusWord : Word;   // Temporary status
                tempWord : Word;   // Temporary word variable
                tempPointer : Int;   // Temporary pointer variable
                tempLoopIndex : Int;   // Temporary loop index variable
                tempBlkVariant : Int;   // Temporary result of MOVE_BLK_VARIANT
                tempCmdStatus : DWord;   // Temporary status of WRREC and RDREC command
                tempDWord : DWord;   // Temporary DWord variable
                tempVoidHeader : LAcycCom_Typestatheader;   // Temporary empty header structure
                tempActualElementReal : LAcycCom_typeDriveDataset;   // Temporary element of the dataset (real values)
             END_VAR
             IF (statrequestBuffer.GetRessource(statAllocatedIndex)=LAcycCom_ResourceManagerRetval#STATUS_BUSY) THEN

                CASE  statFBSubState OF
                    LAcycCom_ReadWriteStatus#FB_GET_SUBSTATE:
                        statFBSubState := LAcycCom_ReadWriteStatus#FB_BUSY_WRREC_1;
                        statReqReadParameter.parameterAddress[0] := statReqParameterInit;
                        FOR tempLoopIndex := 0 TO LENGTH_WRITE_TELEGRAM_UPPER_LIM DO
                           atmpRec[tempLoopIndex] := byte#0;
                        END_FOR;

                    LAcycCom_ReadWriteStatus#FB_BUSY_WRREC_1,  LAcycCom_ReadWriteStatus#FB_BUSY_WRREC_2:  // Writing the dataset configuration into the drive object

                    IF (statCmdBusy = FALSE) AND (statFBSubState =  LAcycCom_ReadWriteStatus#FB_BUSY_WRREC_1) AND  not(statFBState = LAcycCom_ReadWriteStatus#FB_ERROR) THEN
                      // Resets WRREC command
                       instWRREC(request := FALSE,
                                     RECORD := atmpSend);

                      // Creating header data
                       statReqReadParameter.header.refNo :=  statRefNo; // Telegram reference number
                       statReqReadParameter.header.reqId := byte#16#01;  // 0x01 = request parameters
                       statReqReadParameter.header.doId :=  statDoId;  // Drive object identification number
                       statReqReadParameter.header.parameterNo := byte#16#01;  // Count of parameters

                      // Copying the dataset into a static variable
                       statParameter[0].index := uint#0;
                       statParameter[0].parameterNo :=  statParameterNumber;
                       statParameter[0].realValue :=  statParameterValue;
                       statParameter[0].dwordValue := statParameterDWValue;
                       statReqReadParameter.parameterAddress[0].parameterNo :=  statParameter[0].parameterNo;  // Parameter number
                       statReqReadParameter.parameterAddress[0].index :=  statParameter[0].index;  // Subindex of parameter

                    ELSIF (statCmdBusy = FALSE) AND (statFBSubState =  LAcycCom_ReadWriteStatus#FB_BUSY_WRREC_2) AND  not(statFBState = LAcycCom_ReadWriteStatus#FB_ERROR) THEN
                      // Resets WRREC command
                       instWRREC(request := FALSE,
                                     RECORD := atmpSend);

                      // Creating header data
                       statReqWriteParameter.header.refNo :=  statRefNo; // Telegram reference number
                       statReqWriteParameter.header.reqId := byte#16#02;  // 0x02 = change parameters
                       statReqWriteParameter.header.doId :=  statDoId;  // Drive object identification number
                       statReqWriteParameter.header.parameterNo := byte#16#01;  // Count of parameters

                      // Creating parameter address - parameter number and parameter index
                       statReqWriteParameter.data[0] := byte#16#10; // Attribute of parameters (0x10=Value, 0x30=Text)
                       statReqWriteParameter.data[1] := byte#16#01; // No. of elements (for single elements=1)
                       statParameter[0].index :=  statindex;
                       statParameter[0].parameterNo :=  statParameterNumber;

                      // Parameter number
                       statReqWriteParameter.data[3] :=  statParameter[0].parameterNo.%B0;
                       statReqWriteParameter.data[2] :=  statParameter[0].parameterNo.%B1;

                      // Subindex of parameter
                       statReqWriteParameter.data[5] :=  statParameter[0].index.%B0;
                       statReqWriteParameter.data[4] :=  statParameter[0].index.%B1;

                      // Creating parameter address - data
                      IF (statParameter[0].format =  FORMAT_ERROR) THEN
                         statParameter[0].format := TO_BYTE(FORMAT_FLOATING_POINT);
                      END_IF;

                       statReqWriteParameter.data[6] :=  statParameter[0].format; // Format of parameter
                       statReqWriteParameter.data[7] := byte#16#01; // Count of values

                      CASE TO_SINT(statParameter[0].format) OF
                         FORMAT_INTEGER_8:
                          // V1.5.2: Added using of dword value input
                          IF (statParameter[0].realValue = 0.0) THEN
                             tempDWord :=  statParameter[0].dwordValue;
                          ELSE
                             tempDWord := TO_DWORD(TO_SINT(statParameter[0].realValue));
                          END_IF;

                           statReqWriteParameter.data[9] :=  tempDWord.%B1;
                           statReqWriteParameter.data[8] :=  tempDWord.%B0;

                         FORMAT_INTEGER_16:
                          // V1.5.2: Added using of dword value input
                          IF (statParameter[0].realValue = 0.0) THEN
                             tempDWord :=  statParameter[0].dwordValue;
                          ELSE
                             tempDWord := TO_DWORD(TO_DINT(statParameter[0].realValue));
                          END_IF;

                           statReqWriteParameter.data[9] :=  tempDWord.%B0;
                           statReqWriteParameter.data[8] :=  tempDWord.%B1;

                         FORMAT_INTEGER_32:
                          // V1.5.2: Added using of dword value input
                          IF (statParameter[0].realValue = 0.0) THEN
                             tempDWord :=  statParameter[0].dwordValue;
                          ELSE
                             tempDWord := TO_DWORD(TO_DINT(statParameter[0].realValue));
                          END_IF;

                           statReqWriteParameter.data[11] :=  tempDWord.%B0;
                           statReqWriteParameter.data[10] :=  tempDWord.%B1;
                           statReqWriteParameter.data[9] :=  tempDWord.%B2;
                           statReqWriteParameter.data[8] :=  tempDWord.%B3;

                         FORMAT_UNSIGNED_8,  FORMAT_OCTET_STRING: // V1.5 change OCTET_STRING:
                          // V1.5.2: Added using of dword value input
                          IF (statParameter[0].realValue = 0.0) THEN
                             tempDWord :=  statParameter[0].dwordValue;
                          ELSE
                             tempDWord := TO_DWORD(TO_USINT(statParameter[0].realValue));
                          END_IF;

                           statReqWriteParameter.data[9] :=  tempDWord.%B1;
                           statReqWriteParameter.data[8] :=  tempDWord.%B0;

                         FORMAT_UNSIGNED_16:
                          // V1.5.2: Added using of dword value input
                          IF (statParameter[0].realValue = 0.0) THEN
                             tempDWord :=  statParameter[0].dwordValue;
                          ELSE
                             tempDWord := TO_DWORD(TO_UDINT(statParameter[0].realValue));
                          END_IF;

                           statReqWriteParameter.data[9] :=  tempDWord.%B0;
                           statReqWriteParameter.data[8] :=  tempDWord.%B1;

                         FORMAT_UNSIGNED_32,  FORMAT_TIME_DIFFERENCE:
                          // V1.5.2: Added using of dword value input
                          IF (statParameter[0].realValue = 0.0) THEN
                             tempDWord :=  statParameter[0].dwordValue;
                          ELSE
                             tempDWord := TO_DWORD(TO_UDINT(statParameter[0].realValue));
                          END_IF;

                           statReqWriteParameter.data[11] :=  tempDWord.%B0;
                           statReqWriteParameter.data[10] :=  tempDWord.%B1;
                           statReqWriteParameter.data[9] :=  tempDWord.%B2;
                           statReqWriteParameter.data[8] :=  tempDWord.%B3;

                         FORMAT_FLOATING_POINT,  FORMAT_DOUBLE_WORD:
                          // V1.5.2: Added using of dword value input
                          IF (statParameter[0].realValue = 0.0) THEN
                             tempDWord :=  statParameter[0].dwordValue;
                          ELSE
                             tempDWord := TO_DWORD(statParameter[0].realValue);
                          END_IF;

                           statReqWriteParameter.data[11] :=  tempDWord.%B0;
                           statReqWriteParameter.data[10] :=  tempDWord.%B1;
                           statReqWriteParameter.data[9] :=  tempDWord.%B2;
                           statReqWriteParameter.data[8] :=  tempDWord.%B3;

                         FORMAT_BYTE:
                          // V1.5.2: Added using of dword value input
                          IF (statParameter[0].realValue = 0.0) THEN
                             tempDWord :=  statParameter[0].dwordValue;
                          ELSE
                             tempDWord := TO_DWORD(statParameter[0].realValue);
                          END_IF;

                           statReqWriteParameter.data[9] :=  tempDWord.%B1;
                           statReqWriteParameter.data[8] :=  tempDWord.%B0;

                         FORMAT_WORD:
                          // V1.5.2: Added using of dword value input
                          IF (statParameter[0].realValue = 0.0) THEN
                             tempDWord :=  statParameter[0].dwordValue;
                          ELSE
                             tempDWord := TO_DWORD(statParameter[0].realValue);
                          END_IF;

                           statReqWriteParameter.data[9] :=  tempDWord.%B0;
                           statReqWriteParameter.data[8] :=  tempDWord.%B1;

                        ELSE
                          ;
                      END_CASE;
                    END_IF; //  statCmdBusy = FALSE AND  statParameterConfig = TRUE

                    IF (statFBSubState =  LAcycCom_ReadWriteStatus#FB_BUSY_WRREC_1) AND  not(statFBState = LAcycCom_ReadWriteStatus#FB_ERROR) THEN
                      // WRREC command
                                 // Data record
                      SerializeBig(uint#0,
                                     statReqReadParameter,
                                      atmpSend );

                       instWRREC(request := TRUE,                                                // Transfer data record
                                 ID :=  statHwId,                                                // ID number of the hardware component
                                 INDEX :=  statDataRecordNo,                                     // Data record number
                                 LENGTH := uint#0,                                               // Maximum length of the data record to be transferred in bytes
                                 DONE =>  statCmdDone,                                           // Data record was transferred
                                 BUSY =>  statCmdBusy,                                           // The writing process is not yet complete
                                 ERROR =>  statCmdError,                                         // An error occurred during the writing process
                                 STATUS =>  tempCmdStatus,                                       // Status[1] = Error => Status[2] Error Decode + Status[3] Error Code
                                 RECORD :=  atmpSend);                                           // Data record

                                       // Data record

                    ELSIF (statFBSubState =  LAcycCom_ReadWriteStatus#FB_BUSY_WRREC_2) AND  not(statFBState = LAcycCom_ReadWriteStatus#FB_ERROR) THEN
                      // WRREC command
                      SerializeBig(uint#0,
                      statReqWriteParameter,
                      atmpSend );

                       instWRREC(request := TRUE,                                                // Transfer data record
                                 ID :=  statHwId,                                                // ID number of the hardware component
                                 INDEX :=  statDataRecordNo,                                     // Data record number
                                 LENGTH := uint#0,                                               // Maximum length of the data record to be transferred in bytes
                                 DONE =>  statCmdDone,                                           // Data record was transferred
                                 BUSY =>  statCmdBusy,                                           // The writing process is not yet complete
                                 ERROR =>  statCmdError,                                         // An error occurred during the writing process
                                 STATUS =>  tempCmdStatus,                                       // Status[1] = Error => Status[2] Error Decode + Status[3] Error Code
                                 RECORD :=  atmpSend);                                           // Data record
                    END_IF;

                    // Error occurred
                    IF (statCmdError = TRUE) AND  not(statFBState = LAcycCom_ReadWriteStatus#FB_ERROR) THEN
                      // Get the error information from the status information
                       tempStatusWord.%B0 :=  tempCmdStatus.%B1;
                       tempStatusWord.%B1 :=  tempCmdStatus.%B2;

                      // Temporary command status (80A1, 80A7, 80B5, 80C0, 80C1, 80C2, 80C3 oder 80C4) are valid and retry command
                      IF (tempStatusWord = word#16#80A1) OR  // Negative acknowledgment when writing to the module
                        (tempStatusWord = word#16#80A7) OR   // DP slave or module is occupied (temporary error)
                        (tempStatusWord = word#16#80B5) OR   // DP slave or module not ready
                        (tempStatusWord = word#16#80C0) OR   // The data can only be written when the CPU is in STOP mode. Note: this means that writing by the user program is not possible. You can only write the data online with PG/PC.
                        (tempStatusWord = word#16#80C1) OR   // The data of the previous write job on the module for the same data record have not yet been processed by the module.
                        (tempStatusWord = word#16#80C2) OR   // The module is currently processing the maximum possible number of jobs for a CPU.
                        (tempStatusWord = word#16#80C3) OR   // The required operating resources are currently occupied.
                        (tempStatusWord = word#16#80C4) THEN // Internal temporary error. Job could not be executed. Repeat the job. If this error occurs often, check your installation for sources of electrical interference.

                        IF (statErrorCount >=  MAX_ERROR_COUNT) THEN

                           statStateNumber :=  statFBSubState;
                           statSubfunctionStatus :=  tempStatusWord;
                           statStatus :=  ERR_WRREC_TEMP_COUNTER;
                           statFBState :=   LAcycCom_ReadWriteStatus#FB_ERROR;
                        ELSE
                           statErrorCount :=  statErrorCount + usint#1;  // Increment internal error counter
                           statFBSubStateOld :=  statFBSubState;
                           statFBSubState :=  LAcycCom_ReadWriteStatus#FB_BUSY_WAIT;
                        END_IF;
                      ELSE
                         statStateNumber :=  statFBSubState;
                         statSubfunctionStatus :=  tempStatusWord;
                         statStatus :=  ERR_WRREC;
                         statFBState :=   LAcycCom_ReadWriteStatus#FB_ERROR;
                      END_IF; // Temporary command status (80A1, 80A7, 80B5, 80C0, 80C1, 80C2, 80C3 oder 80C4) are valid and retry command

                    ELSIF (statCmdBusy = FALSE) AND (statCmdDone = TRUE) AND  not(statFBState = LAcycCom_ReadWriteStatus#FB_ERROR) AND (statFBSubState =  LAcycCom_ReadWriteStatus#FB_BUSY_WRREC_1) THEN  // Processing completed without errors
                       statErrorCount := uint#0;  // V1.5.1 Reset error counter
                       statFBSubState :=  LAcycCom_ReadWriteStatus#FB_BUSY_RDREC_1; // WRREC completed and continue with RDREC

                    ELSIF (statCmdBusy = FALSE) AND (statCmdDone = TRUE) AND  not(statFBState = LAcycCom_ReadWriteStatus#FB_ERROR) AND (statFBSubState =  LAcycCom_ReadWriteStatus#FB_BUSY_WRREC_2) THEN  // Processing completed without errors
                       statErrorCount := uint#0;  // V1.5.1 Reset error counter
                       statFBSubState :=  LAcycCom_ReadWriteStatus#FB_BUSY_RDREC_2; // WRREC completed and continue with RDREC
                    END_IF; //  statCmdError = TRUE

                    LAcycCom_ReadWriteStatus#FB_BUSY_RDREC_1,  LAcycCom_ReadWriteStatus#FB_BUSY_RDREC_2:  // Reading the values from the drive object

                    // Resets RDREC command
                    IF (statCmdBusy = FALSE) THEN
                       instRDREC(request := FALSE,
                                 RECORD :=  atmpRec);
                    END_IF;

                     instRDREC(request := TRUE,                                                 // Transfer data record
                               ID :=  statHwId,                                                 // ID number of the hardware component
                               INDEX :=  statDataRecordNo,                                                     // Data record number
                               MAXLENGTH := uint#0,                                                       // Maximum length in bytes of the data record information to be read
                               VALID =>  tempCmdValid,                                          // New data record was received and is valid
                               BUSY =>  statCmdBusy,                                            // The reading process is not yet complete
                               ERROR =>  statCmdError,                                          // An error occurred during the reading process
                               STATUS =>  tempCmdStatus,                                        // Status[1] = Error => Status[2] Error Decode + Status[3] Error Code
                               RECORD :=  atmpRec);                                   // Destination area for the data record read

                               DeserializeBig(uint#0,
                               atmpRec,
                               statRespParameter);		                                  // Destination area for the data record read

                    // Error occurred
                    IF (statCmdError = TRUE) AND  not(statFBState = LAcycCom_ReadWriteStatus#FB_ERROR) THEN
                      // Get the error information from the status information
                       tempStatusWord.%B0 :=  tempCmdStatus.%B1;
                       tempStatusWord.%B1 :=  tempCmdStatus.%B2;

                      // Temporary command status (80A0, 80A7, 80B5, 80C0, 80C1, 80C2, 80C3 oder 80C4) are valid and retry command
                      IF (tempStatusWord = word#16#80A0) OR  // Negative acknowledgment when reading the module
                        (tempStatusWord = word#16#80A7) OR   // DP slave or module is occupied (temporary error)
                        (tempStatusWord = word#16#80B5) OR   // DP slave or module not ready
                        (tempStatusWord = word#16#80C0) OR   // The data can only be written when the CPU is in STOP mode. Note: this means that writing by the user program is not possible. You can only write the data online with PG/PC.
                        (tempStatusWord = word#16#80C1) OR   // The data of the previous write job on the module for the same data record have not yet been processed by the module.
                        (tempStatusWord = word#16#80C2) OR   // The module is currently processing the maximum possible number of jobs for a CPU.
                        (tempStatusWord = word#16#80C3) OR   // The required operating resources are currently occupied.
                        (tempStatusWord = word#16#80C4) THEN // Internal temporary error. Job could not be executed. Repeat the job. If this error occurs often, check your installation for sources of electrical interference.

                        IF (statErrorCount >=  MAX_ERROR_COUNT) THEN

                           statStateNumber :=  statFBSubState;
                           statSubfunctionStatus :=  tempStatusWord;
                           statStatus :=  ERR_RDREC_TEMP_COUNTER;
                           statFBState :=   LAcycCom_ReadWriteStatus#FB_ERROR;
                        ELSE
                           statErrorCount :=  statErrorCount + usint#1;  // Increment internal error counter
                           statFBSubStateOld :=  statFBSubState;
                          // V1.3.2. If error 80A0 then should be retry with WRREC command
                          IF (tempStatusWord = word#16#80A0) AND  statFBSubState =  LAcycCom_ReadWriteStatus#FB_BUSY_RDREC_1 THEN
                             statFBSubStateOld :=  LAcycCom_ReadWriteStatus#FB_BUSY_WRREC_1;
                          ELSIF (tempStatusWord = word#16#80A0) AND  statFBSubState =  LAcycCom_ReadWriteStatus#FB_BUSY_RDREC_2 THEN
                             statFBSubStateOld :=  LAcycCom_ReadWriteStatus#FB_BUSY_WRREC_2;
                          END_IF;
                           statFBSubState :=  LAcycCom_ReadWriteStatus#FB_BUSY_WAIT;
                        END_IF;
                      ELSE

                         statStateNumber :=  statFBSubState;
                         statSubfunctionStatus :=  tempStatusWord;
                         statStatus :=  ERR_RDREC;
                         statFBState :=   LAcycCom_ReadWriteStatus#FB_ERROR;
                      END_IF; // Temporary command status (80A0, 80A7, 80B5, 80C0, 80C1, 80C2, 80C3 oder 80C4) are valid and retry command

                      // Error : Reference number of the request does not match with the response reference number
                    ELSIF (statCmdBusy = FALSE) AND
                      (statRefNo <> statRespParameter.header.refNo) AND
                      (tempCmdValid = TRUE) THEN

                       statStateNumber :=  statFBSubState;
                       statStatus :=  ERR_REFERENCE_NO;
                       statFBState :=   LAcycCom_ReadWriteStatus#FB_ERROR;

                      // Error : Invalid response from the drive object (reqId: 16#01 - reading parameter successful; 16#81: reading parameter finished with error; 16#02: writing parameter sucessful; 16#82: writing parameter finished with error)
                    ELSIF (statCmdBusy = FALSE) AND
                      NOT (statRespParameter.header.reqId = byte#16#81 OR  statRespParameter.header.reqId = byte#16#01 OR  statRespParameter.header.reqId = byte#16#02 OR  statRespParameter.header.reqId = byte#16#82) AND
                      (tempCmdValid = TRUE) THEN

                       statStateNumber :=  statFBSubState;
                       statStatus :=  ERR_RESPONSE_ID;
                       statFBState :=   LAcycCom_ReadWriteStatus#FB_ERROR;

                      // Error : The received number of parameters does not match with the requested number of parameters
                    ELSIF (statCmdBusy = FALSE) AND
                      (TO_INT(statRespParameter.header.parameterNo) <> 1) AND
                      (tempCmdValid = TRUE) THEN

                       statStateNumber :=  statFBSubState;
                       statStatus :=  ERR_PARAMETER_NO;
                       statFBState :=   LAcycCom_ReadWriteStatus#FB_ERROR;

                      // Error : The drive object does not match with the responsed DO
                    ELSIF (statCmdBusy = FALSE) AND
                      (statDoId <>  statRespParameter.header.doId) AND
                      (tempCmdValid = TRUE) THEN

                       statStateNumber :=  statFBSubState;
                       statStatus :=  ERR_DRIVE_OBJECT_NO;
                       statFBState :=   LAcycCom_ReadWriteStatus#FB_ERROR;

                      // No error occurred during reading parameters
                    ELSIF (statCmdBusy = FALSE) AND (tempCmdValid = TRUE) AND  not(statFBState = LAcycCom_ReadWriteStatus#FB_ERROR) THEN

                      IF (statFBSubState =  LAcycCom_ReadWriteStatus#FB_BUSY_RDREC_1) THEN

                        // Analyse of the response buffer
                         statParameter[0].format :=  statRespParameter.data[0];  // Format of the parameter

                        // Format = Error
                        IF (((TO_SINT(statRespParameter.data[0]) >  FORMAT_DOUBLE_WORD) OR
                          ((TO_SINT(statRespParameter.data[0]) >  FORMAT_FLOATING_POINT) AND (TO_SINT(statRespParameter.data[0]) <  FORMAT_OCTET_STRING)) OR
                          ((TO_SINT(statRespParameter.data[0]) >  FORMAT_OCTET_STRING) AND (TO_SINT(statRespParameter.data[0]) <  FORMAT_TIME_DIFFERENCE)) OR
                          ((TO_SINT(statRespParameter.data[0]) >  FORMAT_TIME_DIFFERENCE) AND (TO_SINT(statRespParameter.data[0]) <  FORMAT_BYTE)) OR
                          (TO_SINT(statRespParameter.data[0]) <  FORMAT_INTEGER_8))) AND (TO_SINT(statRespParameter.data[0]) <>  FORMAT_ZERO)
                        THEN
                           statParameter[0].errorValue :=  statRespParameter.data[3];

                        ELSE
                           statParameter[0].errorValue := byte#16#FF; // Sets the error status and diagnostic
                           statdiagnostics.errorValue :=  statParameter[0].errorValue;
                        END_IF; // Format = Error

                         statCmdBusy := FALSE;
                         statCmdError := FALSE;
                         statFBState :=  LAcycCom_ReadWriteStatus#FB_BUSY;
                         statFBSubState :=  LAcycCom_ReadWriteStatus#FB_BUSY_WRREC_2;

                      ELSE
                        // Error occurred during writing process (changing parameter values)
                        IF (statRespParameter.header.reqId = byte#16#82) THEN  // reqId: 16#82 (Error occurred during writing paramaters)

                          // Parameter error
                          IF (statRespParameter.data[0] =  FORMAT_ERROR) THEN

                            // Save first parameter error in telegram
                                IF (statFirstParameterError =  NO_PARAMETER_ERROR) THEN
                                statFirstParameterError := 0;
                                statdiagnostics.firstParameterError :=  statFirstParameterError;

                                statStateNumber :=  statFBSubState;
                                statStatus :=  ERR_PARAMETER;
                                statFBState :=   LAcycCom_ReadWriteStatus#FB_ERROR;
                                END_IF;

                             statParameter[0].errorValue :=  statRespParameter.data[3];
                             statdiagnostics.errorValue :=  statParameter[0].errorValue; // V1.3.2

                            // Parameter without errors
                          ELSE
                             statParameter[0].errorValue := byte#16#FF;
                          END_IF;

                          statdiagnostics.errorValue :=  statParameter[0].errorValue;
                        END_IF; // Error occurred during writing process (changing parameter values)

                         statCmdBusy := FALSE;
                         statCmdError := FALSE;
                         statFBSubState :=  LAcycCom_ReadWriteStatus#FB_BUSY_WRREC_1;

                            // Next state is depending on the FB mode
                            IF not(statFBState = LAcycCom_ReadWriteStatus#FB_ERROR) THEN
                                statStatus := STATUS_RELEASE;
                                statFBState := LAcycCom_ReadWriteStatus#FB_RELEASE;

                            END_IF; // statMode = MODE_WITH_BUFFER_MANAGER
                      END_IF; //  statParameterConfig = TRUE
                    END_IF; //  statCmdError = TRUE

                    LAcycCom_ReadWriteStatus#FB_BUSY_WAIT:
                    // Timer for temporary errors
                     instIECTimer(signal :=  statTimerStart,
                                 duration :=  TIMER_TEMP_ERROR);

                     statTimerStart := TRUE;
                    IF (instIECTimer.output = TRUE) THEN
                       statTimerStart := FALSE;
                       statFBSubState :=  statFBSubStateOld;
                    END_IF;

                  ELSE

                     statStatus :=  ERR_UNDEFINED_SUBSTATE;
                     statStateNumber :=  statFBState;
                     statFBState :=   LAcycCom_ReadWriteStatus#FB_ERROR;
                END_CASE;

              ELSE

                 statStatus :=  ERR_COMMAND_TIMEOUT;
                 statStateNumber :=  statFBState;
                 statFBState :=   LAcycCom_ReadWriteStatus#FB_ERROR;
              END_IF; // ((buffer.element[statAllocatedIndex].enable = TRUE) AND (statMode =  MODE_WITH_BUFFER_MANAGER)) OR  statMode =  MODE_WITHOUT_BUFFER_MANAGER

        END_METHOD

        METHOD PUBLIC Start : bool
            VAR_INPUT
                  driveObjectId  : UInt := UINT#0;   // Optional: Identification number of the drive object (value =0: driveObjectId is not used, i.e. the corresponding drive object is only addressed via the hardwareId)
                  hardwareId : HW_IO;   // Hardware identifier of the hardware module
                  parameterNumber : UInt;   // Number of the parameter
                  index : UInt;   // Parameter index
                  value   : REAL;
                  DWVALUE : DWORD;
            END_VAR

             statparameterNumber := parameterNumber;
             statindex := index;
             statParameterValue := value;
             statParameterDWValue := DWVALUE;
             statDoId := to_byte(driveObjectId);
             statHwId := hardwareId;

             // starts functionality
             IF not ((statFBState = LAcycCom_ReadWriteStatus#FB_IDLE OR
                 statFBState = LAcycCom_ReadWriteStatus#FB_DONE) AND
                 statrequestBuffer <> NULL) THEN
                   Start := False;
             ELSE
               // Initialisation
               Start := TRUE;
               statAllocatedIndex := -1;
               statSubfunctionStatus :=  word#16#0000;
               statDataRecordNo := dint#0;
               statStateNumber := LAcycCom_ReadWriteStatus#FB_IDLE;
               statDatasetType := SINT#0;
               statFirstParameterError := -1;
               statErrorCount := uint#0;
               statFBSubState := LAcycCom_ReadWriteStatus#FB_BUSY_WRREC;
               statFBState := LAcycCom_ReadWriteStatus#FB_FIRST_CYCLE;

               instIECTimer(signal := FALSE,
                             duration := TIMER_ALLOCATION);

             END_IF;
        END_METHOD

    END_CLASS
END_NAMESPACE
